// TIA Portal V20 export
DATA_BLOCK "T4 LANT HMI"   // DB1212
{ S7_Optimized_Access := 'TRUE' }
AUTHOR : SAS
// stored: AutoNumber false, IsRetainMemResEnabled true, MemoryReserve 100, RetainMemoryReserve 100
   VAR
      Conditions : Struct
         CG : "Pop_Up_Aux";   // General conditions
         CA : "Pop_Up_Aux";   // Start Auto mode conditions
         SC : "Pop_Up_Aux";   // Start cycle conditions
         MOV_FW_LANT : "Pop_Up_Aux";   // Movement interlocks Forward Lant
         MOV_BW_LANT : "Pop_Up_Aux";   // Movement interlocks Backward Lant
         MOV_FW_LANT_ROST : "Pop_Up_Aux";   // Movement interlocks Forward Lant Rost
         MOV_BW_LANT_ROST : "Pop_Up_Aux";   // Movement interlocks Backward Lant Rost
      END_STRUCT;
      HMI : Struct
         PB : Struct
            s0 : Bool;
            s1 : Bool;
            s2 : Bool;
            s3 : Bool;
            s4 : Bool;
            Pause : Bool;   // Pause
            s6 : Bool;
            s7 : Bool;
            s8 : Bool;
            s9 : Bool;
            s10 : Bool;
            s11 : Bool;
            s12 : Bool;
            s13 : Bool;
            s14 : Bool;
            s15 : Bool;
         END_STRUCT;
         ST : Struct
            s0 : Bool;
            s1 : Bool;
            s2 : Bool;
            s3 : Bool;
            s4 : Bool;
            Pause : Bool;   // Pause
            s6 : Bool;
            s7 : Bool;
            s8 : Bool;
            s9 : Bool;
            "ST Machine" : Int;   // Device label status (0=EME, 1=Safe, 2=Fault, 3=Run, 4=Stopped)
            "ST Sequencer step" : Int;   // Sequencer step
         END_STRUCT;
      END_STRUCT;
   END_VAR
BEGIN
   // Conditions.CG.Conditions.n1 : Tensiune Alimentare OK
   // Conditions.CG.Conditions.n2 : Electric protectie OK
   // Conditions.CG.Conditions.n3 : Inverter OK
   // Conditions.CA.Conditions.n1 : Conditiie Generale
   // Conditions.SC.Conditions.n1 : Initial Conditions
   // Conditions.SC.Conditions.n2 : Piece Presence
   // Conditions.SC.Conditions.n3 : Tracking OK
   // Conditions.SC.Conditions.n4 : Condition of movement
   // Conditions.SC.Conditions.n5 : T4-Exentric
   // Conditions.SC.Conditions.n6 : T4 Opritor
   // Conditions.MOV_FW_LANT.Conditions.n1 : Permanent Conditions
   // Conditions.MOV_BW_LANT.Conditions.n1 : Permanent Conditions
   // Conditions.MOV_BW_LANT.Conditions.n2 : No Teava pe Pozitia Start Bancal
   // Conditions.MOV_FW_LANT_ROST.Conditions.n1 : Permanent Conditions
   // Conditions.MOV_BW_LANT_ROST.Conditions.n1 : Permanent Conditions
   // Conditions.MOV_BW_LANT_ROST.Conditions.n2 : No TimeOut Cuplare/Decupl. Alim.Inv.LantRost
   // Conditions.MOV_BW_LANT_ROST.Conditions.n3 : Sectionator Alim. InvMotLantRost T4-Decuplat
END_DATA_BLOCK
